    movel([0.250450, -0.478284, -2.826261, -1.407844, 1.570796, 1.821246],accel_mss,speed_ms,0,blend_radius_m)
    speed_ms = 0.040
    movel([0.142859, -0.556896, -2.822391, -1.333102, 1.570796, 1.713655],accel_mss,speed_ms,0,blend_radius_m)
    speed_ms = 0.005
    movel([0.142859, -0.561969, -2.829283, -1.321137, 1.570796, 1.713655],accel_mss,speed_ms,0,blend_radius_m)
    speed_ms = 0.025
    movel([0.147960, -0.561530, -2.829311, -1.321548, 1.570796, 1.718757],accel_mss,speed_ms,0,blend_radius_m)
    movel([0.152507, -0.561997, -2.829281, -1.321111, 1.570796, 1.723303],accel_mss,speed_ms,0,blend_radius_m)
    movel([0.156518, -0.563307, -2.829198, -1.319885, 1.570796, 1.727315],accel_mss,speed_ms,0,blend_radius_m)
    movel([0.160009, -0.565397, -2.829063, -1.317930, 1.570796, 1.730805],accel_mss,speed_ms,0,blend_radius_m)
    movel([0.162981, -0.568211, -2.828879, -1.315299, 1.570796, 1.733777],accel_mss,speed_ms,0,blend_radius_m)
    movel([0.165471, -0.571674, -2.828648, -1.312067, 1.570796, 1.736267],accel_mss,speed_ms,0,blend_radius_m)
    movel([0.167478, -0.575738, -2.828372, -1.308279, 1.570796, 1.738275],accel_mss,speed_ms,0,blend_radius_m)
    movel([0.169045, -0.580313, -2.828054, -1.304023, 1.570796, 1.739842],accel_mss,speed_ms,0,blend_radius_m)
    movel([0.170174, -0.585349, -2.827694, -1.299345, 1.570796, 1.740970],accel_mss,speed_ms,0,blend_radius_m)
    movel([0.170906, -0.590770, -2.827297, -1.294322, 1.570796, 1.741702],accel_mss,speed_ms,0,blend_radius_m)
    movel([0.171252, -0.596510, -2.826864, -1.289015, 1.570796, 1.742049],accel_mss,speed_ms,0,blend_radius_m)
    movel([0.171240, -0.602514, -2.826397, -1.283477, 1.570796, 1.742037],accel_mss,speed_ms,0,blend_radius_m)
    movel([0.170896, -0.608698, -2.825903, -1.277789, 1.570796, 1.741692],accel_mss,speed_ms,0,blend_radius_m)
    movel([0.170231, -0.615023, -2.825381, -1.271985, 1.570796, 1.741027],accel_mss,speed_ms,0,blend_radius_m)
    movel([0.169277, -0.621405, -2.824840, -1.266145, 1.570796, 1.740073],accel_mss,speed_ms,0,blend_radius_m)
    movel([0.168058, -0.627794, -2.824281, -1.260314, 1.570796, 1.738854],accel_mss,speed_ms,0,blend_radius_m)
    movel([0.166067, -0.636472, -2.823497, -1.252420, 1.570796, 1.736863],accel_mss,speed_ms,0,blend_radius_m)
    movel([0.163315, -0.646641, -2.822540, -1.243209, 1.570796, 1.734111],accel_mss,speed_ms,0,blend_radius_m)
    movel([0.159729, -0.657566, -2.821465, -1.233358, 1.570796, 1.730525],accel_mss,speed_ms,0,blend_radius_m)
    movel([0.157601, -0.663090, -2.820903, -1.228397, 1.570796, 1.728397],accel_mss,speed_ms,0,blend_radius_m)
    movel([0.155245, -0.668526, -2.820337, -1.223526, 1.570796, 1.726041],accel_mss,speed_ms,0,blend_radius_m)
    movel([0.152635, -0.673812, -2.819775, -1.218802, 1.570796, 1.723431],accel_mss,speed_ms,0,blend_radius_m)
    movel([0.149772, -0.678842, -2.819230, -1.214317, 1.570796, 1.720569],accel_mss,speed_ms,0,blend_radius_m)
    movel([0.146633, -0.683554, -2.818709, -1.210126, 1.570796, 1.717430],accel_mss,speed_ms,0,blend_radius_m)
    movel([0.143204, -0.687871, -2.818224, -1.206294, 1.570796, 1.714001],accel_mss,speed_ms,0,blend_radius_m)
    movel([0.139476, -0.691706, -2.817786, -1.202897, 1.570796, 1.710272],accel_mss,speed_ms,0,blend_radius_m)
    movel([0.135423, -0.695000, -2.817405, -1.199984, 1.570796, 1.706219],accel_mss,speed_ms,0,blend_radius_m)
    movel([0.133263, -0.696421, -2.817239, -1.198729, 1.570796, 1.704059],accel_mss,speed_ms,0,blend_radius_m)
    movel([0.131015, -0.697682, -2.817091, -1.197616, 1.570796, 1.701811],accel_mss,speed_ms,0,blend_radius_m)
    movel([0.126237, -0.699687, -2.816854, -1.195848, 1.570796, 1.697033],accel_mss,speed_ms,0,blend_radius_m)
    movel([0.120774, -0.701207, -2.816674, -1.194508, 1.570796, 1.691570],accel_mss,speed_ms,0,blend_radius_m)
    movel([0.115779, -0.702029, -2.816576, -1.193784, 1.570796, 1.686575],accel_mss,speed_ms,0,blend_radius_m)
    movel([0.111192, -0.702237, -2.816551, -1.193601, 1.570796, 1.681989],accel_mss,speed_ms,0,blend_radius_m)
    movel([0.106936, -0.701901, -2.816591, -1.193896, 1.570796, 1.677733],accel_mss,speed_ms,0,blend_radius_m)
    movel([0.102954, -0.701095, -2.816687, -1.194607, 1.570796, 1.673750],accel_mss,speed_ms,0,blend_radius_m)
    movel([0.099174, -0.699900, -2.816829, -1.195660, 1.570796, 1.669970],accel_mss,speed_ms,0,blend_radius_m)
    movel([0.091955, -0.696634, -2.817214, -1.198541, 1.570796, 1.662751],accel_mss,speed_ms,0,blend_radius_m)
    movel([0.084230, -0.692675, -2.817674, -1.202040, 1.570796, 1.655026],accel_mss,speed_ms,0,blend_radius_m)
    movel([0.076710, -0.688522, -2.818150, -1.205717, 1.570796, 1.647506],accel_mss,speed_ms,0,blend_radius_m)
    movel([0.069639, -0.683747, -2.818688, -1.209954, 1.570796, 1.640435],accel_mss,speed_ms,0,blend_radius_m)
    movel([0.066356, -0.680978, -2.818995, -1.212416, 1.570796, 1.637152],accel_mss,speed_ms,0,blend_radius_m)
    movel([0.063282, -0.677875, -2.819336, -1.215178, 1.570796, 1.634079],accel_mss,speed_ms,0,blend_radius_m)
    movel([0.059324, -0.674172, -2.819737, -1.218480, 1.570796, 1.630120],accel_mss,speed_ms,0,blend_radius_m)
    movel([0.054766, -0.671076, -2.820068, -1.221245, 1.570796, 1.625562],accel_mss,speed_ms,0,blend_radius_m)
    movel([0.049693, -0.668549, -2.820335, -1.223505, 1.570796, 1.620490],accel_mss,speed_ms,0,blend_radius_m)
    movel([0.044211, -0.666515, -2.820548, -1.225326, 1.570796, 1.615008],accel_mss,speed_ms,0,blend_radius_m)
    movel([0.032399, -0.663712, -2.820839, -1.227838, 1.570796, 1.603196],accel_mss,speed_ms,0,blend_radius_m)
    movel([0.020133, -0.662121, -2.821002, -1.229266, 1.570796, 1.590929],accel_mss,speed_ms,0,blend_radius_m)
    movel([0.010394, -0.661823, -2.821033, -1.229534, 1.570796, 1.581190],accel_mss,speed_ms,0,blend_radius_m)
    movel([-0.000051, -0.662753, -2.820937, -1.228699, 1.570796, 1.570745],accel_mss,speed_ms,0,blend_radius_m)
    movel([-0.011149, -0.664929, -2.820713, -1.226747, 1.570796, 1.559647],accel_mss,speed_ms,0,blend_radius_m)
    movel([-0.022832, -0.668377, -2.820353, -1.223659, 1.570796, 1.547964],accel_mss,speed_ms,0,blend_radius_m)
    movel([-0.035034, -0.673085, -2.819853, -1.219451, 1.570796, 1.535762],accel_mss,speed_ms,0,blend_radius_m)
    movel([-0.041303, -0.675912, -2.819549, -1.216928, 1.570796, 1.529494],accel_mss,speed_ms,0,blend_radius_m)
    movel([-0.054134, -0.682501, -2.818826, -1.211062, 1.570796, 1.516662],accel_mss,speed_ms,0,blend_radius_m)
    movel([-0.060678, -0.686261, -2.818406, -1.207722, 1.570796, 1.510118],accel_mss,speed_ms,0,blend_radius_m)
    movel([-0.073954, -0.694686, -2.817441, -1.200262, 1.570796, 1.496842],accel_mss,speed_ms,0,blend_radius_m)
    movel([-0.083094, -0.701206, -2.816674, -1.194509, 1.570796, 1.487702],accel_mss,speed_ms,0,blend_radius_m)
    movel([-0.092241, -0.708453, -2.815799, -1.188136, 1.570796, 1.478555],accel_mss,speed_ms,0,blend_radius_m)
    movel([-0.101295, -0.716344, -2.814820, -1.181225, 1.570796, 1.469501],accel_mss,speed_ms,0,blend_radius_m)
    movel([-0.110164, -0.724811, -2.813739, -1.173839, 1.570796, 1.460632],accel_mss,speed_ms,0,blend_radius_m)
    movel([-0.118767, -0.733783, -2.812558, -1.166048, 1.570796, 1.452030],accel_mss,speed_ms,0,blend_radius_m)
    movel([-0.127013, -0.743184, -2.811280, -1.157925, 1.570796, 1.443783],accel_mss,speed_ms,0,blend_radius_m)
    movel([-0.134825, -0.752948, -2.809910, -1.149532, 1.570796, 1.435971],accel_mss,speed_ms,0,blend_radius_m)
    movel([-0.142128, -0.763002, -2.808451, -1.140936, 1.570796, 1.428668],accel_mss,speed_ms,0,blend_radius_m)
    movel([-0.148437, -0.772501, -2.807028, -1.132859, 1.570796, 1.422359],accel_mss,speed_ms,0,blend_radius_m)
    movel([-0.154044, -0.781724, -2.805605, -1.125060, 1.570796, 1.416752],accel_mss,speed_ms,0,blend_radius_m)
    movel([-0.158917, -0.790659, -2.804185, -1.117545, 1.570796, 1.411879],accel_mss,speed_ms,0,blend_radius_m)
    movel([-0.163027, -0.799306, -2.802773, -1.110310, 1.570796, 1.407769],accel_mss,speed_ms,0,blend_radius_m)
    movel([-0.164788, -0.803524, -2.802070, -1.106795, 1.570796, 1.406008],accel_mss,speed_ms,0,blend_radius_m)
    movel([-0.167695, -0.811728, -2.800677, -1.099984, 1.570796, 1.403101],accel_mss,speed_ms,0,blend_radius_m)
    movel([-0.168834, -0.815720, -2.799987, -1.096683, 1.570796, 1.401963],accel_mss,speed_ms,0,blend_radius_m)
    movel([-0.170468, -0.823474, -2.798621, -1.090294, 1.570796, 1.400328],accel_mss,speed_ms,0,blend_radius_m)
    movel([-0.170957, -0.827243, -2.797946, -1.087201, 1.570796, 1.399840],accel_mss,speed_ms,0,blend_radius_m)
    movel([-0.171222, -0.830932, -2.797277, -1.084180, 1.570796, 1.399575],accel_mss,speed_ms,0,blend_radius_m)
    movel([-0.171271, -0.836014, -2.796344, -1.080031, 1.570796, 1.399525],accel_mss,speed_ms,0,blend_radius_m)
    movel([-0.170997, -0.840889, -2.795436, -1.076064, 1.570796, 1.399800],accel_mss,speed_ms,0,blend_radius_m)
    movel([-0.170424, -0.845545, -2.794557, -1.072288, 1.570796, 1.400372],accel_mss,speed_ms,0,blend_radius_m)
    movel([-0.169586, -0.849986, -2.793706, -1.068697, 1.570796, 1.401210],accel_mss,speed_ms,0,blend_radius_m)
    movel([-0.168498, -0.854186, -2.792892, -1.065311, 1.570796, 1.402298],accel_mss,speed_ms,0,blend_radius_m)
    movel([-0.167183, -0.858136, -2.792117, -1.062136, 1.570796, 1.403613],accel_mss,speed_ms,0,blend_radius_m)
    movel([-0.165667, -0.861831, -2.791384, -1.059174, 1.570796, 1.405129],accel_mss,speed_ms,0,blend_radius_m)
    movel([-0.163968, -0.865252, -2.790699, -1.056439, 1.570796, 1.406828],accel_mss,speed_ms,0,blend_radius_m)
    movel([-0.155842, -0.877159, -2.788259, -1.046970, 1.570796, 1.414954],accel_mss,speed_ms,0,blend_radius_m)
    movel([-0.149559, -0.886895, -2.786203, -1.039291, 1.570796, 1.421237],accel_mss,speed_ms,0,blend_radius_m)
    movel([-0.149099, -0.887946, -2.785978, -1.038465, 1.570796, 1.421697],accel_mss,speed_ms,0,blend_radius_m)
    movel([-0.141673, -0.877908, -2.788103, -1.046377, 1.570796, 1.429123],accel_mss,speed_ms,0,blend_radius_m)
    movel([-0.133733, -0.867970, -2.790149, -1.054270, 1.570796, 1.437064],accel_mss,speed_ms,0,blend_radius_m)
    movel([-0.125327, -0.858167, -2.792111, -1.062111, 1.570796, 1.445469],accel_mss,speed_ms,0,blend_radius_m)
    movel([-0.116525, -0.848549, -2.793983, -1.069857, 1.570796, 1.454272],accel_mss,speed_ms,0,blend_radius_m)
    movel([-0.107391, -0.839172, -2.795758, -1.077460, 1.570796, 1.463405],accel_mss,speed_ms,0,blend_radius_m)
    movel([-0.097997, -0.830079, -2.797432, -1.084877, 1.570796, 1.472800],accel_mss,speed_ms,0,blend_radius_m)
    movel([-0.088413, -0.821332, -2.799001, -1.092056, 1.570796, 1.482383],accel_mss,speed_ms,0,blend_radius_m)
    movel([-0.078723, -0.812984, -2.800461, -1.098944, 1.570796, 1.492073],accel_mss,speed_ms,0,blend_radius_m)
    movel([-0.074112, -0.809252, -2.801101, -1.102035, 1.570796, 1.496684],accel_mss,speed_ms,0,blend_radius_m)
    movel([-0.069384, -0.805683, -2.801707, -1.104999, 1.570796, 1.501412],accel_mss,speed_ms,0,blend_radius_m)
    movel([-0.064581, -0.802315, -2.802273, -1.107801, 1.570796, 1.506215],accel_mss,speed_ms,0,blend_radius_m)
    movel([-0.059754, -0.799201, -2.802790, -1.110398, 1.570796, 1.511043],accel_mss,speed_ms,0,blend_radius_m)
    movel([-0.054946, -0.796380, -2.803255, -1.112754, 1.570796, 1.515851],accel_mss,speed_ms,0,blend_radius_m)
    movel([-0.050200, -0.793899, -2.803660, -1.114830, 1.570796, 1.520596],accel_mss,speed_ms,0,blend_radius_m)
    movel([-0.045567, -0.791799, -2.804001, -1.116589, 1.570796, 1.525229],accel_mss,speed_ms,0,blend_radius_m)
    movel([-0.041096, -0.790126, -2.804271, -1.117992, 1.570796, 1.529701],accel_mss,speed_ms,0,blend_radius_m)
    movel([-0.036831, -0.788923, -2.804464, -1.119002, 1.570796, 1.533966],accel_mss,speed_ms,0,blend_radius_m)
    movel([-0.032817, -0.788231, -2.804575, -1.119583, 1.570796, 1.537980],accel_mss,speed_ms,0,blend_radius_m)
    movel([-0.029108, -0.788094, -2.804597, -1.119698, 1.570796, 1.541689],accel_mss,speed_ms,0,blend_radius_m)
    movel([-0.025747, -0.788549, -2.804524, -1.119316, 1.570796, 1.545049],accel_mss,speed_ms,0,blend_radius_m)
    movel([-0.022782, -0.789633, -2.804350, -1.118406, 1.570796, 1.548014],accel_mss,speed_ms,0,blend_radius_m)
    movel([-0.020249, -0.791380, -2.804069, -1.116940, 1.570796, 1.550547],accel_mss,speed_ms,0,blend_radius_m)
    movel([-0.018198, -0.793823, -2.803673, -1.114893, 1.570796, 1.552598],accel_mss,speed_ms,0,blend_radius_m)
    movel([-0.016670, -0.796996, -2.803154, -1.112239, 1.570796, 1.554126],accel_mss,speed_ms,0,blend_radius_m)
    movel([-0.015425, -0.801968, -2.802331, -1.108090, 1.570796, 1.555371],accel_mss,speed_ms,0,blend_radius_m)
    movel([-0.014861, -0.807651, -2.801374, -1.103364, 1.570796, 1.555935],accel_mss,speed_ms,0,blend_radius_m)
    movel([-0.014879, -0.813881, -2.800306, -1.098203, 1.570796, 1.555917],accel_mss,speed_ms,0,blend_radius_m)
    movel([-0.015374, -0.820500, -2.799149, -1.092741, 1.570796, 1.555423],accel_mss,speed_ms,0,blend_radius_m)
    movel([-0.016250, -0.827353, -2.797926, -1.087111, 1.570796, 1.554546],accel_mss,speed_ms,0,blend_radius_m)
    movel([-0.017417, -0.834297, -2.796661, -1.081431, 1.570796, 1.553380],accel_mss,speed_ms,0,blend_radius_m)
    movel([-0.020226, -0.847879, -2.794111, -1.070399, 1.570796, 1.550570],accel_mss,speed_ms,0,blend_radius_m)
    movel([-0.022367, -0.856502, -2.792439, -1.063448, 1.570796, 1.548430],accel_mss,speed_ms,0,blend_radius_m)
    movel([-0.024863, -0.865087, -2.790732, -1.056570, 1.570796, 1.545933],accel_mss,speed_ms,0,blend_radius_m)
    movel([-0.027666, -0.873630, -2.788991, -1.049768, 1.570796, 1.543130],accel_mss,speed_ms,0,blend_radius_m)
    movel([-0.030732, -0.882151, -2.787212, -1.043026, 1.570796, 1.540064],accel_mss,speed_ms,0,blend_radius_m)
    movel([-0.034013, -0.890645, -2.785396, -1.036348, 1.570796, 1.536783],accel_mss,speed_ms,0,blend_radius_m)
    movel([-0.037464, -0.899123, -2.783539, -1.029726, 1.570796, 1.533332],accel_mss,speed_ms,0,blend_radius_m)
    movel([-0.044724, -0.916079, -2.779693, -1.016617, 1.570796, 1.526072],accel_mss,speed_ms,0,blend_radius_m)
    movel([-0.037887, -0.916184, -2.779669, -1.016536, 1.570796, 1.532909],accel_mss,speed_ms,0,blend_radius_m)
    movel([-0.034369, -0.916506, -2.779594, -1.016289, 1.570796, 1.536427],accel_mss,speed_ms,0,blend_radius_m)
    movel([-0.031381, -0.917369, -2.779393, -1.015627, 1.570796, 1.539415],accel_mss,speed_ms,0,blend_radius_m)
    movel([-0.030227, -0.918088, -2.779225, -1.015075, 1.570796, 1.540569],accel_mss,speed_ms,0,blend_radius_m)
    movel([-0.029375, -0.919046, -2.779002, -1.014342, 1.570796, 1.541421],accel_mss,speed_ms,0,blend_radius_m)
    movel([-0.028875, -0.920267, -2.778715, -1.013407, 1.570796, 1.541921],accel_mss,speed_ms,0,blend_radius_m)
    movel([-0.028783, -0.921786, -2.778358, -1.012245, 1.570796, 1.542014],accel_mss,speed_ms,0,blend_radius_m)
    movel([-0.029151, -0.923626, -2.777923, -1.010840, 1.570796, 1.541646],accel_mss,speed_ms,0,blend_radius_m)
    movel([-0.030036, -0.925829, -2.777399, -1.009161, 1.570796, 1.540761],accel_mss,speed_ms,0,blend_radius_m)
    movel([-0.031485, -0.928421, -2.776779, -1.007189, 1.570796, 1.539311],accel_mss,speed_ms,0,blend_radius_m)
    movel([-0.033550, -0.931424, -2.776055, -1.004910, 1.570796, 1.537247],accel_mss,speed_ms,0,blend_radius_m)
    movel([-0.035465, -0.933874, -2.775460, -1.003055, 1.570796, 1.535331],accel_mss,speed_ms,0,blend_radius_m)
    movel([-0.037392, -0.936083, -2.774920, -1.001386, 1.570796, 1.533404],accel_mss,speed_ms,0,blend_radius_m)
    movel([-0.039326, -0.938069, -2.774432, -0.999888, 1.570796, 1.531471],accel_mss,speed_ms,0,blend_radius_m)
    movel([-0.043222, -0.941457, -2.773593, -0.997339, 1.570796, 1.527575],accel_mss,speed_ms,0,blend_radius_m)
    movel([-0.045180, -0.942896, -2.773235, -0.996258, 1.570796, 1.525616],accel_mss,speed_ms,0,blend_radius_m)
    movel([-0.049122, -0.945366, -2.772616, -0.994407, 1.570796, 1.521674],accel_mss,speed_ms,0,blend_radius_m)
    movel([-0.053080, -0.947408, -2.772102, -0.992879, 1.570796, 1.517716],accel_mss,speed_ms,0,blend_radius_m)
    movel([-0.057051, -0.949170, -2.771655, -0.991564, 1.570796, 1.513746],accel_mss,speed_ms,0,blend_radius_m)
    movel([-0.064972, -0.952410, -2.770829, -0.989150, 1.570796, 1.505824],accel_mss,speed_ms,0,blend_radius_m)
    movel([-0.069092, -0.959193, -2.769076, -0.984119, 1.570796, 1.501705],accel_mss,speed_ms,0,blend_radius_m)
    movel([-0.071347, -0.962585, -2.768188, -0.981616, 1.570796, 1.499449],accel_mss,speed_ms,0,blend_radius_m)
    movel([-0.073742, -0.965885, -2.767316, -0.979188, 1.570796, 1.497055],accel_mss,speed_ms,0,blend_radius_m)
    movel([-0.076282, -0.969024, -2.766480, -0.976886, 1.570796, 1.494514],accel_mss,speed_ms,0,blend_radius_m)
    movel([-0.078972, -0.971932, -2.765699, -0.974759, 1.570796, 1.491824],accel_mss,speed_ms,0,blend_radius_m)
    movel([-0.081818, -0.974540, -2.764993, -0.972856, 1.570796, 1.488978],accel_mss,speed_ms,0,blend_radius_m)
    movel([-0.084835, -0.976790, -2.764380, -0.971219, 1.570796, 1.485961],accel_mss,speed_ms,0,blend_radius_m)
    movel([-0.086956, -0.977940, -2.764066, -0.970384, 1.570796, 1.483841],accel_mss,speed_ms,0,blend_radius_m)
    movel([-0.088635, -0.978358, -2.763951, -0.970080, 1.570796, 1.482161],accel_mss,speed_ms,0,blend_radius_m)
    movel([-0.089921, -0.978151, -2.764008, -0.970230, 1.570796, 1.480875],accel_mss,speed_ms,0,blend_radius_m)
    movel([-0.090856, -0.977421, -2.764208, -0.970760, 1.570796, 1.479941],accel_mss,speed_ms,0,blend_radius_m)
    movel([-0.091484, -0.976268, -2.764523, -0.971598, 1.570796, 1.479312],accel_mss,speed_ms,0,blend_radius_m)
    movel([-0.091845, -0.974803, -2.764921, -0.972664, 1.570796, 1.478951],accel_mss,speed_ms,0,blend_radius_m)
    movel([-0.091988, -0.973126, -2.765376, -0.973887, 1.570796, 1.478808],accel_mss,speed_ms,0,blend_radius_m)
    movel([-0.091944, -0.971335, -2.765859, -0.975195, 1.570796, 1.478853],accel_mss,speed_ms,0,blend_radius_m)
    movel([-0.091464, -0.967350, -2.766926, -0.978112, 1.570796, 1.479332],accel_mss,speed_ms,0,blend_radius_m)
    movel([-0.090613, -0.963214, -2.768022, -0.981152, 1.570796, 1.480183],accel_mss,speed_ms,0,blend_radius_m)
    movel([-0.088355, -0.954571, -2.770274, -0.987543, 1.570796, 1.482442],accel_mss,speed_ms,0,blend_radius_m)
    movel([-0.097400, -0.953356, -2.770587, -0.988447, 1.570796, 1.473396],accel_mss,speed_ms,0,blend_radius_m)
    movel([-0.106686, -0.952546, -2.770794, -0.989049, 1.570796, 1.464111],accel_mss,speed_ms,0,blend_radius_m)
    movel([-0.115967, -0.951708, -2.771009, -0.989673, 1.570796, 1.454830],accel_mss,speed_ms,0,blend_radius_m)
    movel([-0.120533, -0.951142, -2.771153, -0.990094, 1.570796, 1.450264],accel_mss,speed_ms,0,blend_radius_m)
    movel([-0.125013, -0.950404, -2.771341, -0.990643, 1.570796, 1.445784],accel_mss,speed_ms,0,blend_radius_m)
    movel([-0.129176, -0.949478, -2.771577, -0.991334, 1.570796, 1.441621],accel_mss,speed_ms,0,blend_radius_m)
    movel([-0.133191, -0.948361, -2.771861, -0.992168, 1.570796, 1.437605],accel_mss,speed_ms,0,blend_radius_m)
    movel([-0.140952, -0.945765, -2.772516, -0.994108, 1.570796, 1.429844],accel_mss,speed_ms,0,blend_radius_m)
    movel([-0.148657, -0.943103, -2.773183, -0.996103, 1.570796, 1.422140],accel_mss,speed_ms,0,blend_radius_m)
    movel([-0.156652, -0.940856, -2.773743, -0.997790, 1.570796, 1.414144],accel_mss,speed_ms,0,blend_radius_m)
    movel([-0.158404, -0.945856, -2.772493, -0.994040, 1.570796, 1.412393],accel_mss,speed_ms,0,blend_radius_m)
    movel([-0.159893, -0.950717, -2.771262, -0.990410, 1.570796, 1.410903],accel_mss,speed_ms,0,blend_radius_m)
    movel([-0.161122, -0.955430, -2.770053, -0.986906, 1.570796, 1.409674],accel_mss,speed_ms,0,blend_radius_m)
    movel([-0.162097, -0.959989, -2.768869, -0.983531, 1.570796, 1.408699],accel_mss,speed_ms,0,blend_radius_m)
    movel([-0.162817, -0.964392, -2.767711, -0.980285, 1.570796, 1.407979],accel_mss,speed_ms,0,blend_radius_m)
    movel([-0.163294, -0.968633, -2.766584, -0.977172, 1.570796, 1.407503],accel_mss,speed_ms,0,blend_radius_m)
    movel([-0.163522, -0.972706, -2.765490, -0.974194, 1.570796, 1.407274],accel_mss,speed_ms,0,blend_radius_m)
    movel([-0.163516, -0.976612, -2.764429, -0.971348, 1.570796, 1.407280],accel_mss,speed_ms,0,blend_radius_m)
    movel([-0.163271, -0.980342, -2.763405, -0.968641, 1.570796, 1.407525],accel_mss,speed_ms,0,blend_radius_m)
    movel([-0.162789, -0.983889, -2.762423, -0.966077, 1.570796, 1.408007],accel_mss,speed_ms,0,blend_radius_m)
    movel([-0.162081, -0.987259, -2.761481, -0.963648, 1.570796, 1.408715],accel_mss,speed_ms,0,blend_radius_m)
    movel([-0.161148, -0.990441, -2.760585, -0.961363, 1.570796, 1.409648],accel_mss,speed_ms,0,blend_radius_m)
    movel([-0.159985, -0.993426, -2.759737, -0.959226, 1.570796, 1.410811],accel_mss,speed_ms,0,blend_radius_m)
    movel([-0.158604, -0.996222, -2.758937, -0.957231, 1.570796, 1.412193],accel_mss,speed_ms,0,blend_radius_m)
    movel([-0.157003, -0.998816, -2.758189, -0.955385, 1.570796, 1.413793],accel_mss,speed_ms,0,blend_radius_m)
    movel([-0.155183, -1.001206, -2.757495, -0.953688, 1.570796, 1.415613],accel_mss,speed_ms,0,blend_radius_m)
    movel([-0.151979, -1.004496, -2.756534, -0.951359, 1.570796, 1.418818],accel_mss,speed_ms,0,blend_radius_m)
    movel([-0.148396, -1.007285, -2.755713, -0.949392, 1.570796, 1.422400],accel_mss,speed_ms,0,blend_radius_m)
    movel([-0.144485, -1.009627, -2.755018, -0.947744, 1.570796, 1.426312],accel_mss,speed_ms,0,blend_radius_m)
    movel([-0.140276, -1.011565, -2.754440, -0.946383, 1.570796, 1.430521],accel_mss,speed_ms,0,blend_radius_m)
    movel([-0.135817, -1.013151, -2.753966, -0.945272, 1.570796, 1.434980],accel_mss,speed_ms,0,blend_radius_m)
    movel([-0.131147, -1.014425, -2.753583, -0.944381, 1.570796, 1.439649],accel_mss,speed_ms,0,blend_radius_m)
    movel([-0.126309, -1.015437, -2.753278, -0.943674, 1.570796, 1.444488],accel_mss,speed_ms,0,blend_radius_m)
    movel([-0.121334, -1.016217, -2.753042, -0.943130, 1.570796, 1.449463],accel_mss,speed_ms,0,blend_radius_m)
    movel([-0.111086, -1.017328, -2.752705, -0.942355, 1.570796, 1.459710],accel_mss,speed_ms,0,blend_radius_m)
    movel([-0.100706, -1.018189, -2.752444, -0.941756, 1.570796, 1.470090],accel_mss,speed_ms,0,blend_radius_m)
    movel([-0.092837, -1.019132, -2.752157, -0.941100, 1.570796, 1.477960],accel_mss,speed_ms,0,blend_radius_m)
    movel([-0.090127, -1.019243, -2.752123, -0.941023, 1.570796, 1.480669],accel_mss,speed_ms,0,blend_radius_m)
    movel([-0.085238, -1.019024, -2.752190, -0.941175, 1.570796, 1.485559],accel_mss,speed_ms,0,blend_radius_m)
    movel([-0.084217, -1.019182, -2.752142, -0.941065, 1.570796, 1.486579],accel_mss,speed_ms,0,blend_radius_m)
    movel([-0.083300, -1.019548, -2.752030, -0.940811, 1.570796, 1.487496],accel_mss,speed_ms,0,blend_radius_m)
    movel([-0.082505, -1.020188, -2.751835, -0.940366, 1.570796, 1.488292],accel_mss,speed_ms,0,blend_radius_m)
    movel([-0.081849, -1.021166, -2.751536, -0.939687, 1.570796, 1.488947],accel_mss,speed_ms,0,blend_radius_m)
    movel([-0.081367, -1.022553, -2.751110, -0.938726, 1.570796, 1.489429],accel_mss,speed_ms,0,blend_radius_m)
    movel([-0.081196, -1.024133, -2.750624, -0.937632, 1.570796, 1.489600],accel_mss,speed_ms,0,blend_radius_m)
    movel([-0.081306, -1.025872, -2.750086, -0.936431, 1.570796, 1.489490],accel_mss,speed_ms,0,blend_radius_m)
    movel([-0.081672, -1.027751, -2.749502, -0.935136, 1.570796, 1.489125],accel_mss,speed_ms,0,blend_radius_m)
    movel([-0.082267, -1.029736, -2.748882, -0.933771, 1.570796, 1.488530],accel_mss,speed_ms,0,blend_radius_m)
    movel([-0.084046, -1.033940, -2.747559, -0.930890, 1.570796, 1.486750],accel_mss,speed_ms,0,blend_radius_m)
    movel([-0.085182, -1.036105, -2.746873, -0.929412, 1.570796, 1.485615],accel_mss,speed_ms,0,blend_radius_m)
    movel([-0.087804, -1.040436, -2.745487, -0.926466, 1.570796, 1.482993],accel_mss,speed_ms,0,blend_radius_m)
    movel([-0.090749, -1.044616, -2.744136, -0.923637, 1.570796, 1.480048],accel_mss,speed_ms,0,blend_radius_m)
    movel([-0.093814, -1.048453, -2.742883, -0.921053, 1.570796, 1.476982],accel_mss,speed_ms,0,blend_radius_m)
    movel([-0.096822, -1.051771, -2.741789, -0.918829, 1.570796, 1.473974],accel_mss,speed_ms,0,blend_radius_m)
    movel([-0.101532, -1.056269, -2.740293, -0.915827, 1.570796, 1.469264],accel_mss,speed_ms,0,blend_radius_m)
    movel([-0.103973, -1.058358, -2.739592, -0.914439, 1.570796, 1.466823],accel_mss,speed_ms,0,blend_radius_m)
    movel([-0.106452, -1.060327, -2.738927, -0.913134, 1.570796, 1.464344],accel_mss,speed_ms,0,blend_radius_m)
    movel([-0.111501, -1.063907, -2.737712, -0.910770, 1.570796, 1.459296],accel_mss,speed_ms,0,blend_radius_m)
    movel([-0.116596, -1.066975, -2.736662, -0.908753, 1.570796, 1.454201],accel_mss,speed_ms,0,blend_radius_m)
    movel([-0.121663, -1.069492, -2.735794, -0.907104, 1.570796, 1.449133],accel_mss,speed_ms,0,blend_radius_m)
    movel([-0.126616, -1.071419, -2.735125, -0.905844, 1.570796, 1.444181],accel_mss,speed_ms,0,blend_radius_m)
    movel([-0.129028, -1.072148, -2.734872, -0.905369, 1.570796, 1.441768],accel_mss,speed_ms,0,blend_radius_m)
    movel([-0.133676, -1.073116, -2.734535, -0.904738, 1.570796, 1.437120],accel_mss,speed_ms,0,blend_radius_m)
    movel([-0.135892, -1.073341, -2.734456, -0.904592, 1.570796, 1.434904],accel_mss,speed_ms,0,blend_radius_m)
    movel([-0.138706, -1.073384, -2.734441, -0.904564, 1.570796, 1.432090],accel_mss,speed_ms,0,blend_radius_m)
    movel([-0.141382, -1.073174, -2.734515, -0.904701, 1.570796, 1.429414],accel_mss,speed_ms,0,blend_radius_m)
    movel([-0.143932, -1.072741, -2.734666, -0.904983, 1.570796, 1.426864],accel_mss,speed_ms,0,blend_radius_m)
    movel([-0.146378, -1.072125, -2.734880, -0.905384, 1.570796, 1.424418],accel_mss,speed_ms,0,blend_radius_m)
    movel([-0.151023, -1.070475, -2.735453, -0.906460, 1.570796, 1.419774],accel_mss,speed_ms,0,blend_radius_m)
    movel([-0.155449, -1.068501, -2.736136, -0.907752, 1.570796, 1.415347],accel_mss,speed_ms,0,blend_radius_m)
    movel([-0.160830, -1.065792, -2.737068, -0.909530, 1.570796, 1.409966],accel_mss,speed_ms,0,blend_radius_m)
    movel([-0.166031, -1.062765, -2.738101, -0.911523, 1.570796, 1.404766],accel_mss,speed_ms,0,blend_radius_m)
    movel([-0.171006, -1.059397, -2.739242, -0.913750, 1.570796, 1.399790],accel_mss,speed_ms,0,blend_radius_m)
    movel([-0.175718, -1.055670, -2.740493, -0.916226, 1.570796, 1.395078],accel_mss,speed_ms,0,blend_radius_m)
    movel([-0.180121, -1.051552, -2.741862, -0.918975, 1.570796, 1.390676],accel_mss,speed_ms,0,blend_radius_m)
    movel([-0.184164, -1.047018, -2.743353, -0.922018, 1.570796, 1.386633],accel_mss,speed_ms,0,blend_radius_m)
    movel([-0.187804, -1.042041, -2.744970, -0.925378, 1.570796, 1.382992],accel_mss,speed_ms,0,blend_radius_m)
    movel([-0.190994, -1.036590, -2.746718, -0.929081, 1.570796, 1.379803],accel_mss,speed_ms,0,blend_radius_m)
    movel([-0.193088, -1.032176, -2.748116, -0.932097, 1.570796, 1.377708],accel_mss,speed_ms,0,blend_radius_m)
    movel([-0.195001, -1.027347, -2.749628, -0.935414, 1.570796, 1.375795],accel_mss,speed_ms,0,blend_radius_m)
    movel([-0.196660, -1.022127, -2.751241, -0.939021, 1.570796, 1.374136],accel_mss,speed_ms,0,blend_radius_m)
    movel([-0.197995, -1.016552, -2.752941, -0.942897, 1.570796, 1.372801],accel_mss,speed_ms,0,blend_radius_m)
    movel([-0.198928, -1.010648, -2.754714, -0.947027, 1.570796, 1.371869],accel_mss,speed_ms,0,blend_radius_m)
    movel([-0.199378, -1.004447, -2.756548, -0.951394, 1.570796, 1.371419],accel_mss,speed_ms,0,blend_radius_m)
    movel([-0.199270, -0.997974, -2.758432, -0.955983, 1.570796, 1.371526],accel_mss,speed_ms,0,blend_radius_m)
    movel([-0.198978, -0.994643, -2.759389, -0.958357, 1.570796, 1.371818],accel_mss,speed_ms,0,blend_radius_m)
    movel([-0.198516, -0.991258, -2.760353, -0.960778, 1.570796, 1.372280],accel_mss,speed_ms,0,blend_radius_m)
    movel([-0.197257, -0.984717, -2.762193, -0.965480, 1.570796, 1.373540],accel_mss,speed_ms,0,blend_radius_m)
    movel([-0.195559, -0.977938, -2.764066, -0.970385, 1.570796, 1.375238],accel_mss,speed_ms,0,blend_radius_m)
    movel([-0.193420, -0.970942, -2.765965, -0.975482, 1.570796, 1.377376],accel_mss,speed_ms,0,blend_radius_m)
    movel([-0.190851, -0.963755, -2.767880, -0.980754, 1.570796, 1.379945],accel_mss,speed_ms,0,blend_radius_m)
    movel([-0.187843, -0.956396, -2.769803, -0.986190, 1.570796, 1.382954],accel_mss,speed_ms,0,blend_radius_m)
    movel([-0.184409, -0.948900, -2.771724, -0.991765, 1.570796, 1.386387],accel_mss,speed_ms,0,blend_radius_m)
    movel([-0.180547, -0.941289, -2.773635, -0.997465, 1.570796, 1.390249],accel_mss,speed_ms,0,blend_radius_m)
    movel([-0.176259, -0.933597, -2.775528, -1.003265, 1.570796, 1.394537],accel_mss,speed_ms,0,blend_radius_m)
    movel([-0.185534, -0.925976, -2.777364, -1.009049, 1.570796, 1.385263],accel_mss,speed_ms,0,blend_radius_m)
    movel([-0.190231, -0.922204, -2.778259, -1.011925, 1.570796, 1.380565],accel_mss,speed_ms,0,blend_radius_m)
    movel([-0.194708, -0.918130, -2.779216, -1.015043, 1.570796, 1.376089],accel_mss,speed_ms,0,blend_radius_m)
    movel([-0.197696, -0.914658, -2.780023, -1.017709, 1.570796, 1.373100],accel_mss,speed_ms,0,blend_radius_m)
    movel([-0.200252, -0.910681, -2.780937, -1.020771, 1.570796, 1.370544],accel_mss,speed_ms,0,blend_radius_m)
    movel([-0.202391, -0.906234, -2.781948, -1.024207, 1.570796, 1.368405],accel_mss,speed_ms,0,blend_radius_m)
    movel([-0.204120, -0.901334, -2.783048, -1.028007, 1.570796, 1.366676],accel_mss,speed_ms,0,blend_radius_m)
    movel([-0.205450, -0.896011, -2.784226, -1.032152, 1.570796, 1.365347],accel_mss,speed_ms,0,blend_radius_m)
    movel([-0.206384, -0.890288, -2.785473, -1.036628, 1.570796, 1.364412],accel_mss,speed_ms,0,blend_radius_m)
    movel([-0.206934, -0.884188, -2.786781, -1.041421, 1.570796, 1.363862],accel_mss,speed_ms,0,blend_radius_m)
    movel([-0.207107, -0.877741, -2.788138, -1.046510, 1.570796, 1.363690],accel_mss,speed_ms,0,blend_radius_m)
    movel([-0.206906, -0.870974, -2.789537, -1.051878, 1.570796, 1.363891],accel_mss,speed_ms,0,blend_radius_m)
    movel([-0.206337, -0.863907, -2.790969, -1.057513, 1.570796, 1.364460],accel_mss,speed_ms,0,blend_radius_m)
    movel([-0.205406, -0.856571, -2.792425, -1.063393, 1.570796, 1.365390],accel_mss,speed_ms,0,blend_radius_m)
    movel([-0.204124, -0.848998, -2.793896, -1.069494, 1.570796, 1.366673],accel_mss,speed_ms,0,blend_radius_m)
    movel([-0.202492, -0.841217, -2.795375, -1.075797, 1.570796, 1.368304],accel_mss,speed_ms,0,blend_radius_m)
    movel([-0.200525, -0.833269, -2.796850, -1.082270, 1.570796, 1.370271],accel_mss,speed_ms,0,blend_radius_m)
    movel([-0.198219, -0.825174, -2.798317, -1.088898, 1.570796, 1.372578],accel_mss,speed_ms,0,blend_radius_m)
    movel([-0.195592, -0.816978, -2.799767, -1.095644, 1.570796, 1.375204],accel_mss,speed_ms,0,blend_radius_m)
    movel([-0.189981, -0.801241, -2.802452, -1.108696, 1.570796, 1.380815],accel_mss,speed_ms,0,blend_radius_m)
    movel([-0.186803, -0.793132, -2.803785, -1.115472, 1.570796, 1.383993],accel_mss,speed_ms,0,blend_radius_m)
    movel([-0.183317, -0.784864, -2.805110, -1.122415, 1.570796, 1.387480],accel_mss,speed_ms,0,blend_radius_m)
    movel([-0.179464, -0.776444, -2.806425, -1.129520, 1.570796, 1.391333],accel_mss,speed_ms,0,blend_radius_m)
    movel([-0.175202, -0.767884, -2.807725, -1.136779, 1.570796, 1.395595],accel_mss,speed_ms,0,blend_radius_m)
    movel([-0.170478, -0.759186, -2.809010, -1.144192, 1.570796, 1.400319],accel_mss,speed_ms,0,blend_radius_m)
    movel([-0.165237, -0.750359, -2.810277, -1.151752, 1.570796, 1.405559],accel_mss,speed_ms,0,blend_radius_m)
    movel([-0.158854, -0.740458, -2.811655, -1.160276, 1.570796, 1.411942],accel_mss,speed_ms,0,blend_radius_m)
    movel([-0.151964, -0.730499, -2.812994, -1.168896, 1.570796, 1.418832],accel_mss,speed_ms,0,blend_radius_m)
    movel([-0.144605, -0.720514, -2.814292, -1.177583, 1.570796, 1.426192],accel_mss,speed_ms,0,blend_radius_m)
    movel([-0.136807, -0.710544, -2.815543, -1.186303, 1.570796, 1.433990],accel_mss,speed_ms,0,blend_radius_m)
    movel([-0.128612, -0.700632, -2.816742, -1.195014, 1.570796, 1.442185],accel_mss,speed_ms,0,blend_radius_m)
    movel([-0.120063, -0.690826, -2.817887, -1.203676, 1.570796, 1.450734],accel_mss,speed_ms,0,blend_radius_m)
    movel([-0.111195, -0.681164, -2.818974, -1.212250, 1.570796, 1.459601],accel_mss,speed_ms,0,blend_radius_m)
    movel([-0.102063, -0.671703, -2.820001, -1.220685, 1.570796, 1.468733],accel_mss,speed_ms,0,blend_radius_m)
    movel([-0.092713, -0.662494, -2.820964, -1.228931, 1.570796, 1.478083],accel_mss,speed_ms,0,blend_radius_m)
    movel([-0.083207, -0.653590, -2.821862, -1.236937, 1.570796, 1.487589],accel_mss,speed_ms,0,blend_radius_m)
    movel([-0.073590, -0.645045, -2.822693, -1.244651, 1.570796, 1.497206],accel_mss,speed_ms,0,blend_radius_m)
    movel([-0.063922, -0.636913, -2.823456, -1.252020, 1.570796, 1.506874],accel_mss,speed_ms,0,blend_radius_m)
    movel([-0.054273, -0.629256, -2.824151, -1.258981, 1.570796, 1.516523],accel_mss,speed_ms,0,blend_radius_m)
    movel([-0.044696, -0.622124, -2.824778, -1.265488, 1.570796, 1.526101],accel_mss,speed_ms,0,blend_radius_m)
    movel([-0.035256, -0.615574, -2.825335, -1.271480, 1.570796, 1.535540],accel_mss,speed_ms,0,blend_radius_m)
    movel([-0.026016, -0.609663, -2.825824, -1.276902, 1.570796, 1.544780],accel_mss,speed_ms,0,blend_radius_m)
    movel([-0.016339, -0.603900, -2.826288, -1.282201, 1.570796, 1.554457],accel_mss,speed_ms,0,blend_radius_m)
    movel([-0.006761, -0.598574, -2.826705, -1.287110, 1.570796, 1.564035],accel_mss,speed_ms,0,blend_radius_m)
    movel([0.002637, -0.593828, -2.827068, -1.291493, 1.570796, 1.573433],accel_mss,speed_ms,0,blend_radius_m)
    movel([0.011767, -0.589825, -2.827367, -1.295197, 1.570796, 1.582563],accel_mss,speed_ms,0,blend_radius_m)
    movel([0.022013, -0.586222, -2.827631, -1.298536, 1.570796, 1.592809],accel_mss,speed_ms,0,blend_radius_m)
    movel([0.031836, -0.583741, -2.827810, -1.300838, 1.570796, 1.602632],accel_mss,speed_ms,0,blend_radius_m)
    movel([0.041123, -0.582407, -2.827905, -1.302076, 1.570796, 1.611920],accel_mss,speed_ms,0,blend_radius_m)
    movel([0.049765, -0.582239, -2.827917, -1.302233, 1.570796, 1.620561],accel_mss,speed_ms,0,blend_radius_m)
    movel([0.057667, -0.583237, -2.827846, -1.301306, 1.570796, 1.628463],accel_mss,speed_ms,0,blend_radius_m)
    movel([0.064734, -0.585399, -2.827691, -1.299299, 1.570796, 1.635530],accel_mss,speed_ms,0,blend_radius_m)
    movel([0.070889, -0.588701, -2.827450, -1.296238, 1.570796, 1.641685],accel_mss,speed_ms,0,blend_radius_m)
    movel([0.076060, -0.593121, -2.827121, -1.292147, 1.570796, 1.646856],accel_mss,speed_ms,0,blend_radius_m)
    movel([0.085031, -0.603310, -2.826334, -1.282744, 1.570796, 1.655828],accel_mss,speed_ms,0,blend_radius_m)
    movel([0.088978, -0.608964, -2.825881, -1.277544, 1.570796, 1.659774],accel_mss,speed_ms,0,blend_radius_m)
    movel([0.092366, -0.615396, -2.825350, -1.271643, 1.570796, 1.663163],accel_mss,speed_ms,0,blend_radius_m)
    movel([0.097727, -0.626605, -2.824386, -1.261397, 1.570796, 1.668523],accel_mss,speed_ms,0,blend_radius_m)
    movel([0.100814, -0.631855, -2.823918, -1.256616, 1.570796, 1.671610],accel_mss,speed_ms,0,blend_radius_m)
    movel([0.104295, -0.636627, -2.823483, -1.252279, 1.570796, 1.675092],accel_mss,speed_ms,0,blend_radius_m)
    movel([0.108284, -0.640736, -2.823101, -1.248552, 1.570796, 1.679080],accel_mss,speed_ms,0,blend_radius_m)
    movel([0.112860, -0.644013, -2.822791, -1.245585, 1.570796, 1.683656],accel_mss,speed_ms,0,blend_radius_m)
    movel([0.118142, -0.646276, -2.822575, -1.243538, 1.570796, 1.688938],accel_mss,speed_ms,0,blend_radius_m)
    movel([0.124222, -0.647349, -2.822472, -1.242568, 1.570796, 1.695018],accel_mss,speed_ms,0,blend_radius_m)
    movel([0.126967, -0.647294, -2.822477, -1.242618, 1.570796, 1.697764],accel_mss,speed_ms,0,blend_radius_m)
    movel([0.130048, -0.646603, -2.822544, -1.243243, 1.570796, 1.700844],accel_mss,speed_ms,0,blend_radius_m)
    movel([0.131705, -0.645921, -2.822609, -1.243859, 1.570796, 1.702502],accel_mss,speed_ms,0,blend_radius_m)
    movel([0.133432, -0.644972, -2.822700, -1.244717, 1.570796, 1.704228],accel_mss,speed_ms,0,blend_radius_m)
    movel([0.135229, -0.643713, -2.822820, -1.245856, 1.570796, 1.706025],accel_mss,speed_ms,0,blend_radius_m)
    movel([0.137083, -0.642103, -2.822972, -1.247314, 1.570796, 1.707880],accel_mss,speed_ms,0,blend_radius_m)
    movel([0.138966, -0.640144, -2.823156, -1.249088, 1.570796, 1.709762],accel_mss,speed_ms,0,blend_radius_m)
    movel([0.140743, -0.637984, -2.823357, -1.251048, 1.570796, 1.711539],accel_mss,speed_ms,0,blend_radius_m)
    movel([0.143949, -0.633341, -2.823783, -1.255264, 1.570796, 1.714746],accel_mss,speed_ms,0,blend_radius_m)
    movel([0.145899, -0.630044, -2.824081, -1.258264, 1.570796, 1.716695],accel_mss,speed_ms,0,blend_radius_m)
    movel([0.147600, -0.626796, -2.824370, -1.261224, 1.570796, 1.718397],accel_mss,speed_ms,0,blend_radius_m)
    movel([0.150320, -0.620470, -2.824920, -1.266999, 1.570796, 1.721116],accel_mss,speed_ms,0,blend_radius_m)
    movel([0.152211, -0.614417, -2.825432, -1.272540, 1.570796, 1.723007],accel_mss,speed_ms,0,blend_radius_m)
    movel([0.153394, -0.608671, -2.825905, -1.277813, 1.570796, 1.724190],accel_mss,speed_ms,0,blend_radius_m)
    movel([0.153974, -0.603294, -2.826336, -1.282760, 1.570796, 1.724770],accel_mss,speed_ms,0,blend_radius_m)
    movel([0.154069, -0.598322, -2.826724, -1.287343, 1.570796, 1.724866],accel_mss,speed_ms,0,blend_radius_m)
    movel([0.153795, -0.593802, -2.827070, -1.291518, 1.570796, 1.724591],accel_mss,speed_ms,0,blend_radius_m)
    movel([0.152349, -0.585561, -2.827679, -1.299149, 1.570796, 1.723145],accel_mss,speed_ms,0,blend_radius_m)
    movel([0.151014, -0.581758, -2.827951, -1.302679, 1.570796, 1.721811],accel_mss,speed_ms,0,blend_radius_m)
    movel([0.149274, -0.578388, -2.828188, -1.305812, 1.570796, 1.720070],accel_mss,speed_ms,0,blend_radius_m)
    movel([0.147124, -0.575489, -2.828389, -1.308511, 1.570796, 1.717920],accel_mss,speed_ms,0,blend_radius_m)
    movel([0.144565, -0.573074, -2.828554, -1.310762, 1.570796, 1.715361],accel_mss,speed_ms,0,blend_radius_m)
    movel([0.141602, -0.571175, -2.828682, -1.312532, 1.570796, 1.712399],accel_mss,speed_ms,0,blend_radius_m)
    movel([0.138250, -0.569801, -2.828773, -1.313814, 1.570796, 1.709047],accel_mss,speed_ms,0,blend_radius_m)
    movel([0.134507, -0.568979, -2.828828, -1.314582, 1.570796, 1.705303],accel_mss,speed_ms,0,blend_radius_m)
    speed_ms = 0.005
    movel([0.134507, -0.563781, -2.821946, -1.326663, 1.570796, 1.705303],accel_mss,speed_ms,0,blend_radius_m)
    speed_ms = 0.040
    movel([0.130779, -0.603383, -2.819034, -1.289971, 1.570796, 1.701576],accel_mss,speed_ms,0,blend_radius_m)
    speed_ms = 0.005
    movel([0.130779, -0.609278, -2.825855, -1.277255, 1.570796, 1.701576],accel_mss,speed_ms,0,blend_radius_m)
    speed_ms = 0.025
    movel([0.126088, -0.608692, -2.825903, -1.277794, 1.570796, 1.696885],accel_mss,speed_ms,0,blend_radius_m)
    movel([0.120796, -0.609075, -2.825872, -1.277442, 1.570796, 1.691593],accel_mss,speed_ms,0,blend_radius_m)
    movel([0.117867, -0.609831, -2.825810, -1.276748, 1.570796, 1.688663],accel_mss,speed_ms,0,blend_radius_m)
    movel([0.114729, -0.611066, -2.825709, -1.275614, 1.570796, 1.685525],accel_mss,speed_ms,0,blend_radius_m)
    movel([0.111366, -0.612853, -2.825562, -1.273974, 1.570796, 1.682162],accel_mss,speed_ms,0,blend_radius_m)
    movel([0.107759, -0.615263, -2.825361, -1.271765, 1.570796, 1.678555],accel_mss,speed_ms,0,blend_radius_m)
    speed_ms = 0.005
    movel([0.107759, -0.609268, -2.818550, -1.284570, 1.570796, 1.678555],accel_mss,speed_ms,0,blend_radius_m)
    speed_ms = 0.040
    movel([0.119155, -0.592873, -2.819865, -1.299650, 1.570796, 1.689951],accel_mss,speed_ms,0,blend_radius_m)
    speed_ms = 0.005
    movel([0.119155, -0.598587, -2.826704, -1.287098, 1.570796, 1.689951],accel_mss,speed_ms,0,blend_radius_m)
    speed_ms = 0.025
    movel([0.119329, -0.593456, -2.827096, -1.291838, 1.570796, 1.690125],accel_mss,speed_ms,0,blend_radius_m)
    movel([0.118427, -0.589414, -2.827397, -1.295578, 1.570796, 1.689224],accel_mss,speed_ms,0,blend_radius_m)
    movel([0.116524, -0.586492, -2.827611, -1.298286, 1.570796, 1.687320],accel_mss,speed_ms,0,blend_radius_m)
    movel([0.113681, -0.584752, -2.827737, -1.299900, 1.570796, 1.684478],accel_mss,speed_ms,0,blend_radius_m)
    movel([0.109980, -0.584227, -2.827775, -1.300387, 1.570796, 1.680776],accel_mss,speed_ms,0,blend_radius_m)
    movel([0.105512, -0.584949, -2.827723, -1.299716, 1.570796, 1.676308],accel_mss,speed_ms,0,blend_radius_m)
    movel([0.100370, -0.586937, -2.827579, -1.297873, 1.570796, 1.671167],accel_mss,speed_ms,0,blend_radius_m)
    movel([0.097573, -0.588417, -2.827471, -1.296502, 1.570796, 1.668370],accel_mss,speed_ms,0,blend_radius_m)
    movel([0.094649, -0.590209, -2.827338, -1.294842, 1.570796, 1.665446],accel_mss,speed_ms,0,blend_radius_m)
    speed_ms = 0.005
    movel([0.094649, -0.584638, -2.820487, -1.307264, 1.570796, 1.665446],accel_mss,speed_ms,0,blend_radius_m)
    speed_ms = 0.040
    movel([0.109146, -0.567705, -2.821684, -1.323000, 1.570796, 1.679942],accel_mss,speed_ms,0,blend_radius_m)
    speed_ms = 0.005
    movel([0.109146, -0.572975, -2.828560, -1.310854, 1.570796, 1.679942],accel_mss,speed_ms,0,blend_radius_m)
    speed_ms = 0.025
    movel([0.108766, -0.570826, -2.828705, -1.312858, 1.570796, 1.679563],accel_mss,speed_ms,0,blend_radius_m)
    movel([0.108038, -0.568982, -2.828828, -1.314579, 1.570796, 1.678834],accel_mss,speed_ms,0,blend_radius_m)
    movel([0.105619, -0.566217, -2.829009, -1.317162, 1.570796, 1.676415],accel_mss,speed_ms,0,blend_radius_m)
    movel([0.102068, -0.564691, -2.829108, -1.318589, 1.570796, 1.672864],accel_mss,speed_ms,0,blend_radius_m)
    movel([0.097581, -0.564412, -2.829127, -1.318850, 1.570796, 1.668377],accel_mss,speed_ms,0,blend_radius_m)
    movel([0.092352, -0.565359, -2.829065, -1.317965, 1.570796, 1.663149],accel_mss,speed_ms,0,blend_radius_m)
    movel([0.086610, -0.567499, -2.828926, -1.315965, 1.570796, 1.657407],accel_mss,speed_ms,0,blend_radius_m)
    movel([0.083608, -0.569014, -2.828826, -1.314549, 1.570796, 1.654404],accel_mss,speed_ms,0,blend_radius_m)
    movel([0.077492, -0.572885, -2.828566, -1.310937, 1.570796, 1.648288],accel_mss,speed_ms,0,blend_radius_m)
    movel([0.074432, -0.575231, -2.828407, -1.308752, 1.570796, 1.645229],accel_mss,speed_ms,0,blend_radius_m)
    speed_ms = 0.005
    movel([0.074432, -0.569921, -2.821533, -1.320935, 1.570796, 1.645229],accel_mss,speed_ms,0,blend_radius_m)
    speed_ms = 0.040
    movel([0.095097, -0.548053, -2.822938, -1.341398, 1.570796, 1.665893],accel_mss,speed_ms,0,blend_radius_m)
    speed_ms = 0.005
    movel([0.095097, -0.552964, -2.829841, -1.329584, 1.570796, 1.665893],accel_mss,speed_ms,0,blend_radius_m)
    speed_ms = 0.025
    movel([0.091437, -0.550821, -2.829970, -1.331598, 1.570796, 1.662233],accel_mss,speed_ms,0,blend_radius_m)
    movel([0.086902, -0.549876, -2.830026, -1.332487, 1.570796, 1.657698],accel_mss,speed_ms,0,blend_radius_m)
    movel([0.081586, -0.550188, -2.830008, -1.332194, 1.570796, 1.652383],accel_mss,speed_ms,0,blend_radius_m)
    movel([0.075565, -0.551796, -2.829912, -1.330681, 1.570796, 1.646362],accel_mss,speed_ms,0,blend_radius_m)
    movel([0.068945, -0.554742, -2.829734, -1.327913, 1.570796, 1.639741],accel_mss,speed_ms,0,blend_radius_m)
    movel([0.065442, -0.556721, -2.829612, -1.326056, 1.570796, 1.636238],accel_mss,speed_ms,0,blend_radius_m)
    movel([0.061833, -0.559040, -2.829468, -1.323881, 1.570796, 1.632630],accel_mss,speed_ms,0,blend_radius_m)
    movel([0.058123, -0.561706, -2.829300, -1.321383, 1.570796, 1.628919],accel_mss,speed_ms,0,blend_radius_m)
    movel([0.054326, -0.564721, -2.829107, -1.318562, 1.570796, 1.625123],accel_mss,speed_ms,0,blend_radius_m)
    movel([0.050467, -0.568073, -2.828888, -1.315428, 1.570796, 1.621264],accel_mss,speed_ms,0,blend_radius_m)
    movel([0.046556, -0.571769, -2.828642, -1.311978, 1.570796, 1.617352],accel_mss,speed_ms,0,blend_radius_m)
    speed_ms = 0.005
    movel([0.046556, -0.566521, -2.821763, -1.324104, 1.570796, 1.617352],accel_mss,speed_ms,0,blend_radius_m)
    speed_ms = 0.040
    movel([0.068450, -0.540347, -2.823391, -1.348651, 1.570796, 1.639247],accel_mss,speed_ms,0,blend_radius_m)
    speed_ms = 0.005
    movel([0.068450, -0.545115, -2.830304, -1.336970, 1.570796, 1.639247],accel_mss,speed_ms,0,blend_radius_m)
    speed_ms = 0.025
    movel([0.067250, -0.542563, -2.830450, -1.339377, 1.570796, 1.638046],accel_mss,speed_ms,0,blend_radius_m)
    movel([0.065416, -0.540743, -2.830552, -1.341094, 1.570796, 1.636213],accel_mss,speed_ms,0,blend_radius_m)
    movel([0.062980, -0.539696, -2.830611, -1.342082, 1.570796, 1.633776],accel_mss,speed_ms,0,blend_radius_m)
    movel([0.059988, -0.539453, -2.830624, -1.342312, 1.570796, 1.630785],accel_mss,speed_ms,0,blend_radius_m)
    movel([0.055747, -0.540188, -2.830583, -1.341618, 1.570796, 1.626544],accel_mss,speed_ms,0,blend_radius_m)
    movel([0.051028, -0.541798, -2.830493, -1.340098, 1.570796, 1.621825],accel_mss,speed_ms,0,blend_radius_m)
    movel([0.045096, -0.544498, -2.830339, -1.337551, 1.570796, 1.615893],accel_mss,speed_ms,0,blend_radius_m)
    movel([0.038836, -0.548053, -2.830134, -1.334202, 1.570796, 1.609632],accel_mss,speed_ms,0,blend_radius_m)
    movel([0.032339, -0.552481, -2.829871, -1.330037, 1.570796, 1.603135],accel_mss,speed_ms,0,blend_radius_m)
    movel([0.025694, -0.557813, -2.829544, -1.325032, 1.570796, 1.596490],accel_mss,speed_ms,0,blend_radius_m)
    movel([0.019022, -0.564049, -2.829150, -1.319190, 1.570796, 1.589818],accel_mss,speed_ms,0,blend_radius_m)
    movel([0.015751, -0.567455, -2.828928, -1.316005, 1.570796, 1.586547],accel_mss,speed_ms,0,blend_radius_m)
    movel([0.009514, -0.574699, -2.828443, -1.309247, 1.570796, 1.580311],accel_mss,speed_ms,0,blend_radius_m)
    movel([0.006609, -0.578475, -2.828182, -1.305732, 1.570796, 1.577405],accel_mss,speed_ms,0,blend_radius_m)
    movel([0.003896, -0.582315, -2.827912, -1.302162, 1.570796, 1.574692],accel_mss,speed_ms,0,blend_radius_m)
    movel([0.001401, -0.586195, -2.827633, -1.298561, 1.570796, 1.572197],accel_mss,speed_ms,0,blend_radius_m)
    speed_ms = 0.005
    movel([0.001401, -0.580694, -2.820775, -1.310919, 1.570796, 1.572197],accel_mss,speed_ms,0,blend_radius_m)
    speed_ms = 0.040
    movel([0.024158, -0.545562, -2.823087, -1.343740, 1.570796, 1.594955],accel_mss,speed_ms,0,blend_radius_m)
    speed_ms = 0.005
    movel([0.024158, -0.550426, -2.829993, -1.331969, 1.570796, 1.594955],accel_mss,speed_ms,0,blend_radius_m)
    speed_ms = 0.025
    movel([0.016377, -0.554411, -2.829754, -1.328224, 1.570796, 1.587173],accel_mss,speed_ms,0,blend_radius_m)
    movel([0.008119, -0.559479, -2.829440, -1.323469, 1.570796, 1.578916],accel_mss,speed_ms,0,blend_radius_m)
    movel([-0.000392, -0.565584, -2.829051, -1.317755, 1.570796, 1.570405],accel_mss,speed_ms,0,blend_radius_m)
    movel([-0.004672, -0.569000, -2.828827, -1.314563, 1.570796, 1.566125],accel_mss,speed_ms,0,blend_radius_m)
    movel([-0.008933, -0.572654, -2.828582, -1.311153, 1.570796, 1.561863],accel_mss,speed_ms,0,blend_radius_m)
    movel([-0.013140, -0.576529, -2.828317, -1.307543, 1.570796, 1.557656],accel_mss,speed_ms,0,blend_radius_m)
    movel([-0.017263, -0.580612, -2.828033, -1.303745, 1.570796, 1.553533],accel_mss,speed_ms,0,blend_radius_m)
    movel([-0.021281, -0.584900, -2.827727, -1.299762, 1.570796, 1.549515],accel_mss,speed_ms,0,blend_radius_m)
    movel([-0.025165, -0.589388, -2.827399, -1.295602, 1.570796, 1.545631],accel_mss,speed_ms,0,blend_radius_m)
    movel([-0.028893, -0.594062, -2.827050, -1.291277, 1.570796, 1.541903],accel_mss,speed_ms,0,blend_radius_m)
    movel([-0.032426, -0.598909, -2.826679, -1.286801, 1.570796, 1.538370],accel_mss,speed_ms,0,blend_radius_m)
    movel([-0.035750, -0.603925, -2.826286, -1.282179, 1.570796, 1.535046],accel_mss,speed_ms,0,blend_radius_m)
    movel([-0.038833, -0.609100, -2.825870, -1.277419, 1.570796, 1.531963],accel_mss,speed_ms,0,blend_radius_m)
    speed_ms = 0.005
    movel([-0.038833, -0.603209, -2.819049, -1.290132, 1.570796, 1.531963],accel_mss,speed_ms,0,blend_radius_m)
    speed_ms = 0.040
    movel([-0.023556, -0.569200, -2.821582, -1.321607, 1.570796, 1.547240],accel_mss,speed_ms,0,blend_radius_m)
    speed_ms = 0.005
    movel([-0.023556, -0.574496, -2.828457, -1.309436, 1.570796, 1.547240],accel_mss,speed_ms,0,blend_radius_m)
    speed_ms = 0.025
    movel([-0.027512, -0.576838, -2.828296, -1.307255, 1.570796, 1.543284],accel_mss,speed_ms,0,blend_radius_m)
    movel([-0.031583, -0.579598, -2.828104, -1.304687, 1.570796, 1.539213],accel_mss,speed_ms,0,blend_radius_m)
    movel([-0.035719, -0.582743, -2.827881, -1.301765, 1.570796, 1.535077],accel_mss,speed_ms,0,blend_radius_m)
    movel([-0.039883, -0.586229, -2.827630, -1.298530, 1.570796, 1.530914],accel_mss,speed_ms,0,blend_radius_m)
    movel([-0.044038, -0.590026, -2.827352, -1.295011, 1.570796, 1.526759],accel_mss,speed_ms,0,blend_radius_m)
    movel([-0.048136, -0.594093, -2.827048, -1.291248, 1.570796, 1.522661],accel_mss,speed_ms,0,blend_radius_m)
    movel([-0.052136, -0.598386, -2.826719, -1.287284, 1.570796, 1.518660],accel_mss,speed_ms,0,blend_radius_m)
    movel([-0.056011, -0.602880, -2.826368, -1.283140, 1.570796, 1.514785],accel_mss,speed_ms,0,blend_radius_m)
    movel([-0.059710, -0.607528, -2.825997, -1.278864, 1.570796, 1.511086],accel_mss,speed_ms,0,blend_radius_m)
    movel([-0.063202, -0.612277, -2.825610, -1.274503, 1.570796, 1.507594],accel_mss,speed_ms,0,blend_radius_m)
    movel([-0.066459, -0.617078, -2.825209, -1.270102, 1.570796, 1.504337],accel_mss,speed_ms,0,blend_radius_m)
    movel([-0.069459, -0.621895, -2.824797, -1.265697, 1.570796, 1.501337],accel_mss,speed_ms,0,blend_radius_m)
    movel([-0.072183, -0.626681, -2.824380, -1.261329, 1.570796, 1.498613],accel_mss,speed_ms,0,blend_radius_m)
    movel([-0.074610, -0.631405, -2.823959, -1.257025, 1.570796, 1.496186],accel_mss,speed_ms,0,blend_radius_m)
    movel([-0.076704, -0.636008, -2.823540, -1.252841, 1.570796, 1.494092],accel_mss,speed_ms,0,blend_radius_m)
    movel([-0.078460, -0.640464, -2.823126, -1.248799, 1.570796, 1.492336],accel_mss,speed_ms,0,blend_radius_m)
    speed_ms = 0.005
    movel([-0.078460, -0.634061, -2.816360, -1.261968, 1.570796, 1.492336],accel_mss,speed_ms,0,blend_radius_m)
    speed_ms = 0.040
    movel([-0.070919, -0.605759, -2.818841, -1.287790, 1.570796, 1.499877],accel_mss,speed_ms,0,blend_radius_m)
    speed_ms = 0.005
    movel([-0.070919, -0.611694, -2.825658, -1.275038, 1.570796, 1.499877],accel_mss,speed_ms,0,blend_radius_m)
    speed_ms = 0.025
    movel([-0.074708, -0.614184, -2.825451, -1.272753, 1.570796, 1.496088],accel_mss,speed_ms,0,blend_radius_m)
    movel([-0.078565, -0.617290, -2.825191, -1.269908, 1.570796, 1.492231],accel_mss,speed_ms,0,blend_radius_m)
    movel([-0.082419, -0.620904, -2.824883, -1.266603, 1.570796, 1.488378],accel_mss,speed_ms,0,blend_radius_m)
    movel([-0.086227, -0.624922, -2.824534, -1.262933, 1.570796, 1.484569],accel_mss,speed_ms,0,blend_radius_m)
    movel([-0.089936, -0.629246, -2.824152, -1.258991, 1.570796, 1.480860],accel_mss,speed_ms,0,blend_radius_m)
    movel([-0.093490, -0.633769, -2.823745, -1.254875, 1.570796, 1.477307],accel_mss,speed_ms,0,blend_radius_m)
    movel([-0.096851, -0.638396, -2.823319, -1.250674, 1.570796, 1.473946],accel_mss,speed_ms,0,blend_radius_m)
    movel([-0.099960, -0.643027, -2.822885, -1.246477, 1.570796, 1.470836],accel_mss,speed_ms,0,blend_radius_m)
    movel([-0.102926, -0.647792, -2.822429, -1.242168, 1.570796, 1.467870],accel_mss,speed_ms,0,blend_radius_m)
    movel([-0.105650, -0.652557, -2.821964, -1.237869, 1.570796, 1.465146],accel_mss,speed_ms,0,blend_radius_m)
    movel([-0.108089, -0.657263, -2.821495, -1.233631, 1.570796, 1.462707],accel_mss,speed_ms,0,blend_radius_m)
    movel([-0.110174, -0.661835, -2.821032, -1.229523, 1.570796, 1.460622],accel_mss,speed_ms,0,blend_radius_m)
    movel([-0.111862, -0.666205, -2.820580, -1.225604, 1.570796, 1.458935],accel_mss,speed_ms,0,blend_radius_m)
    movel([-0.113103, -0.670312, -2.820149, -1.221929, 1.570796, 1.457693],accel_mss,speed_ms,0,blend_radius_m)
    movel([-0.113832, -0.674084, -2.819746, -1.218559, 1.570796, 1.456964],accel_mss,speed_ms,0,blend_radius_m)
    movel([-0.114014, -0.677465, -2.819380, -1.215544, 1.570796, 1.456782],accel_mss,speed_ms,0,blend_radius_m)
    speed_ms = 0.005
    movel([-0.114014, -0.670495, -2.812689, -1.229206, 1.570796, 1.456782],accel_mss,speed_ms,0,blend_radius_m)
    speed_ms = 0.040
    movel([-0.116650, -0.652734, -2.814547, -1.245107, 1.570796, 1.454146],accel_mss,speed_ms,0,blend_radius_m)
    speed_ms = 0.005
    movel([-0.116650, -0.659433, -2.821276, -1.231680, 1.570796, 1.454146],accel_mss,speed_ms,0,blend_radius_m)
    speed_ms = 0.025
    movel([-0.121647, -0.665131, -2.820692, -1.226567, 1.570796, 1.449149],accel_mss,speed_ms,0,blend_radius_m)
    movel([-0.126640, -0.671460, -2.820027, -1.220902, 1.570796, 1.444156],accel_mss,speed_ms,0,blend_radius_m)
    movel([-0.131349, -0.678118, -2.819309, -1.214962, 1.570796, 1.439447],accel_mss,speed_ms,0,blend_radius_m)
    movel([-0.135500, -0.684808, -2.818569, -1.209012, 1.570796, 1.435296],accel_mss,speed_ms,0,blend_radius_m)
    movel([-0.138841, -0.691250, -2.817838, -1.203301, 1.570796, 1.431955],accel_mss,speed_ms,0,blend_radius_m)
    movel([-0.140131, -0.694297, -2.817487, -1.200605, 1.570796, 1.430665],accel_mss,speed_ms,0,blend_radius_m)
    movel([-0.141122, -0.697177, -2.817150, -1.198062, 1.570796, 1.429674],accel_mss,speed_ms,0,blend_radius_m)
    movel([-0.141790, -0.699869, -2.816833, -1.195687, 1.570796, 1.429006],accel_mss,speed_ms,0,blend_radius_m)
    movel([-0.142107, -0.702337, -2.816539, -1.193513, 1.570796, 1.428689],accel_mss,speed_ms,0,blend_radius_m)
    movel([-0.142033, -0.704540, -2.816274, -1.191574, 1.570796, 1.428764],accel_mss,speed_ms,0,blend_radius_m)
    movel([-0.141548, -0.706465, -2.816042, -1.189883, 1.570796, 1.429248],accel_mss,speed_ms,0,blend_radius_m)
    speed_ms = 0.005
    movel([-0.141548, -0.699080, -2.809415, -1.203894, 1.570796, 1.429248],accel_mss,speed_ms,0,blend_radius_m)
    speed_ms = 0.040
    movel([-0.150955, -0.698491, -2.809486, -1.204412, 1.570796, 1.419842],accel_mss,speed_ms,0,blend_radius_m)
    speed_ms = 0.005
    movel([-0.150955, -0.705867, -2.816114, -1.190408, 1.570796, 1.419842],accel_mss,speed_ms,0,blend_radius_m)
    speed_ms = 0.025
    movel([-0.156280, -0.715124, -2.814974, -1.182292, 1.570796, 1.414517],accel_mss,speed_ms,0,blend_radius_m)
    movel([-0.158650, -0.719740, -2.814390, -1.178258, 1.570796, 1.412147],accel_mss,speed_ms,0,blend_radius_m)
    movel([-0.160704, -0.724236, -2.813813, -1.174340, 1.570796, 1.410093],accel_mss,speed_ms,0,blend_radius_m)
    movel([-0.162353, -0.728544, -2.813252, -1.170593, 1.570796, 1.408444],accel_mss,speed_ms,0,blend_radius_m)
    movel([-0.163518, -0.732596, -2.812716, -1.167077, 1.570796, 1.407279],accel_mss,speed_ms,0,blend_radius_m)
    movel([-0.164104, -0.736312, -2.812218, -1.163859, 1.570796, 1.406692],accel_mss,speed_ms,0,blend_radius_m)
    movel([-0.164040, -0.739638, -2.811767, -1.160985, 1.570796, 1.406757],accel_mss,speed_ms,0,blend_radius_m)
    speed_ms = 0.005
    movel([-0.164040, -0.704337, -2.778889, -1.229163, 1.570796, 1.406757],accel_mss,speed_ms,0,blend_radius_m)
    speed_ms = 1.000
    movel([-0.164040, -0.704337, -2.778889, -1.229163, 1.570796, 1.406757],accel_mss,speed_ms,0,blend_radius_m)
    # Splitting Linear movement in 6 (instruction 3389: MoveL 3112)
    movel([-0.164040, -0.681322, -2.751226, -1.279841, 1.570796, 1.406757],accel_mss,speed_ms,0,blend_radius_m)
    movel([-0.164040, -0.663017, -2.723351, -1.326021, 1.570796, 1.406757],accel_mss,speed_ms,0,blend_radius_m)
    movel([-0.164040, -0.648620, -2.695283, -1.368486, 1.570796, 1.406757],accel_mss,speed_ms,0,blend_radius_m)
    movel([-0.164040, -0.637500, -2.667032, -1.407857, 1.570796, 1.406757],accel_mss,speed_ms,0,blend_radius_m)
    movel([-0.164040, -0.629153, -2.638608, -1.444627, 1.570796, 1.406757],accel_mss,speed_ms,0,blend_radius_m)
    movel([-0.164040, -0.623175, -2.610015, -1.479199, 1.570796, 1.406757],accel_mss,speed_ms,0,blend_radius_m)
    # End of main program
  end

  Machining1()
  $ 3 "Script: test_second_drawing_8_m18.script"
  def Machining2():
    # Default parameters:
    global speed_ms = 0.3
    global speed_rads = 0.75
    global accel_mss = 3
    global accel_radss = 1.2
    global blend_radius_m = 0.001

